FUNCTION_BLOCK Door (* Template for a simple Basic Function Block Type *)
  (* Standard: 61499-2 *)
  (* Version 1.0, 2019-05-07, jetbrains *)
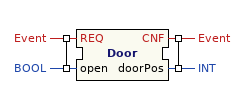
  EVENT_INPUT
    REQ WITH open; (* Normal Execution Request *)
  END_EVENT
  EVENT_OUTPUT
    CNF WITH doorPos; (* Execution Confirmation *)
  END_EVENT
  VAR_INPUT
    open : BOOL; (* Input event qualifier *)
  END_VAR
  VAR_OUTPUT
    doorPos : INT; (* Output event qualifier *)
  END_VAR
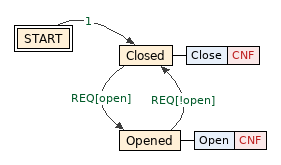
  EC_STATES
    START; (* Initial State *)
    Opened : Open -> CNF;
    Closed : Close -> CNF;
  END_STATES
  EC_TRANSITIONS
    START TO Closed := 1;
    Closed TO Opened := REQ[open];
    Opened TO Closed := REQ[!open];
  END_TRANSITIONS
  ALGORITHM Open IN ST: (* new algorithm *)
doorPos := 10;
  END_ALGORITHM
  ALGORITHM Close IN ST: (* new algorithm *)
doorPos := 0;
  END_ALGORITHM
END_FUNCTION_BLOCK
